FUNCTION_BLOCK FB_AutomaticExtractionStateMachine
VAR_INPUT
	parameters : ST_AutomaticExtractionParameters;
	reactorPressure : DINT;
END_VAR
VAR_OUTPUT
	controlValveOpeningPercentage : DINT;
	decreasePumpSetpoint : BOOL;
	extractivePumpOn : BOOL;
	co2onOffValveClosed : BOOL;
	fillingActive : BOOL;
END_VAR
VAR
	step : INT;
	TON_FillingTimer : TON;
	TON_WaitForValve : TON;
	TON_WaitForPressure : TON;
	TON_KeepExtractivePumpOn : TON;
	startingReactorPRessure : DINT;
END_VAR

CASE step OF 
	
	0: // Extraction step
		IF controlValveOpeningPercentage <> parameters.controlValveOpeningValue THEN
			step := 6;
		END_IF
		fillingActive := FALSE;
		// Start filling timer. When filling timer exceeded, move to filling step
		TON_FillingTimer(
						IN := TRUE,
						PT := TO_TIME(parameters.fillingTime*1000));
		IF TON_FillingTimer.Q THEN
			TON_FillingTimer(IN := FALSE);
			step := step + 1;
		END_IF
	
	1: // Filling step: Control valve to a small opening
		
		fillingActive := TRUE;
		controlValveOpeningPercentage := 20;
		TON_WaitForValve(
						IN := TRUE,
						PT := T#10S);
		IF TON_WaitForValve.Q THEN
			TON_WaitForValve(IN := FALSE);
			step := step + 1;
		END_IF
	
	2: // Set pump setpoint 40 bars lower from current
	
		decreasePumpSetpoint := TRUE;
		TON_WaitForPressure(
							IN := TRUE,
							PT := TO_TIME(parameters.pumpSetpointWaitTime*1000));
		IF TON_WaitForPressure.Q THEN
			TON_WaitForPressure(IN := FALSE);
			step := step + 1;
		END_IF
	
	3: // Close co2 on/off valve, extractive pump on: stays on for a desired time
	
		co2onOffValveClosed := TRUE;
		startingReactorPressure := reactorPressure;
		extractivePumpOn := TRUE;
		TON_KeepExtractivePumpOn(
								IN := TRUE,
								PT := TO_TIME(parameters.pumpOnTime*1000));
		IF TON_KeepExtractivePumpOn.Q THEN
			TON_KeepExtractivePumpOn(IN := FALSE);
			step := step + 1;
		END_IF
	
	4: // Extractive pump turns off after pressure reaches the same as it was b4 turning on
	
		IF startingReactorPRessure = reactorPressure THEN
			extractivePumpOn := FALSE;
			step := step + 1;
		END_IF
		
	5: // Pressure setpoint back to original (+40bar) and open on/off valve
	
		co2onOffValveClosed := FALSE;
		decreasePumpSetpoint := FALSE;
		step := step + 1;
	
	6: // open control valve to desired value
	
		controlValveOpeningPercentage := parameters.controlValveOpeningValue;
		step := 0;
		
END_CASE

METHOD resetState : BOOL
VAR_INPUT
END_VAR

step := 0;
TON_FillingTimer(IN :=FALSE);
TON_WaitForValve(IN :=FALSE);
TON_WaitForPressure(IN :=FALSE);
TON_KeepExtractivePumpOn(IN :=FALSE);
co2onOffValveClosed := FALSE;
decreasePumpSetpoint := FALSE;
extractivePumpOn := FALSE;
fillingActive := FALSE;
END_METHOD

END_FUNCTION_BLOCK

(* stored: Version 1.1.0.1, ProductVersion 3.1.4024.9
   POU FB_AutomaticExtractionStateMachine: Id {fd3c0490-089c-4717-a34f-489c595512a4}, SpecialFunc None
   Method resetState: Id {bf1ce1ba-fd70-4c2a-963b-7e4edcae03f9} *)
